// TIA Portal V19 export
TYPE "C401_VAR_IF_RSS_TYPIC"
   STRUCT
      STS { ExternalAccessible := 'False'; ExternalVisible := 'False'; ExternalWritable := 'False'} : String[8];   // Naam van de getoonde beeldstand (bitmap) op het bord
      EXT_AUT { ExternalAccessible := 'False'; ExternalVisible := 'False'; ExternalWritable := 'False'} : Bool;   // Externe (hoofd) beveiliging aangesproken
      EXT_HW { ExternalAccessible := 'False'; ExternalVisible := 'False'; ExternalWritable := 'False'} : Bool;   // Sturings hardware (PLC) in storing
      STO { ExternalAccessible := 'False'; ExternalVisible := 'False'; ExternalWritable := 'False'} : Struct   // Opsomming van alle storingen en meldingen
         A001 : Bool;   // Beveiliging aangesproken
         A002 : Bool;   // Storing luspaar
         A003 : Bool;   // Storing RSS-bord gedetecteerd door PRTG
         A004 : Bool;   // Storing RSS-bord
         A005 : Bool;   // Algemene storing RSS-bord
      END_STRUCT;
   END_STRUCT;
END_TYPE
